	fbSdoReadExUint		:	FB_EcCoESdoReadEx	:= (bCompleteAccess := FALSE);
	fbSdoReadExUdint	:	FB_EcCoESdoReadEx	:= (bCompleteAccess := FALSE);
	fbSdoWriteExSint		:	FB_EcCoESdoWriteEx 	:= (bCompleteAccess := FALSE);
	fbSdoWriteExInt		:	FB_EcCoESdoWriteEx 	:= (bCompleteAccess := FALSE);
	fbSdoWriteExDint		:	FB_EcCoESdoWriteEx 	:= (bCompleteAccess := FALSE);
	fbSdoWriteExUsint	:	FB_EcCoESdoWriteEx 	:= (bCompleteAccess := FALSE);
	fbSdoWriteExUint		:	FB_EcCoESdoWriteEx 	:= (bCompleteAccess := FALSE);
	fbSdoWriteExUdint	:	FB_EcCoESdoWriteEx 	:= (bCompleteAccess := FALSE);
	fbSdoWriteExString	:	FB_EcCoESdoWriteEx 	:= (bCompleteAccess := FALSE);
	fbEcGetSlaveState	:	FB_EcGetSlaveState		;

	fbFileOpen			:	FB_FileOpen				;	(*Used to determine if file exists*)
	fbFileClose			:	FB_FileClose				;	(*Used to determine if file exists*)
END_VAR

fbFallingEdge	(CLK:= bExecute);
IF fbFallingEdge.Q THEN
	bNotExecute	:=	TRUE;
END_IF;

(* Done is TRUE for one cycle when falling edge of Execute has occured *)
IF bDone AND bNotExecute THEN
	bDone		:=	FALSE;
END_IF;

IF bError AND bNotExecute THEN
	bError				:=	FALSE;
	nErrorId				:=	0;
	nErrorIDRead			:=	0;
END_IF;

CASE State OF
0:
fbRisingEdge(CLK:= bExecute);
IF fbRisingEdge.Q THEN
	bDone				:=	FALSE;
	bBusy				:=	TRUE;
	bError				:=	FALSE;
	nErrorId				:=	0;
	nErrorIDRead			:=	0;
	sErrorString			:=	'';
	bNotExecute			:=	FALSE;
	sNetIdRead			:=	sNetId;
	nSlaveAddrRead		:=	nSlaveAddr;
	sFileRead			:=	sFile;
	bBypassCheckRead	:=	bBypassCheck;
	State				:=	1;
	Row					:=	1;
END_IF

1: (*check if file exists by trying to open the file*)
fbFileOpen(
	nMode		:=	FOPEN_MODEREAD,
	sPathName	:=	sFileRead,
	bExecute	:=	TRUE);
State:=2;

2:
fbFileOpen();
IF NOT fbFileOpen.bBusy THEN			(*Check for File Open complete*)
	IF fbFileOpen.bError THEN			(*Check for error from File Open*)
		sErrorString:=CONCAT(CONCAT(
			'Error opening File at  ',
			sFileRead),
			'.  Error occurred using Function Block FB_FileOpen.  ErrorID is from FB_FileOpen.'
		);
		nErrorIDRead:=fbFileOpen.nErrID;
		State:=99;
	ELSE
		fbFileOpen(bExecute := FALSE);
		fbFileClose(
			hFile		:=fbFileOpen.hFile,
			bExecute	:=TRUE);
		State:=3;
	END_IF
END_IF

3:
fbFileClose();
IF NOT fbFileClose.bBusy THEN			(*Check for File Open complete*)
	IF fbFileClose.bError THEN			(*Check for error from File Open*)
		sErrorString:=CONCAT(CONCAT(
			'Error closing File at  ',
			sFileRead),
			'.  Error occurred using Function Block FB_FileClose.  ErrorID is from FB_FileClose.'
		);
		nErrorIDRead:=fbFileOpen.nErrID;
		State:=99;
	ELSE
		fbFileClose(bExecute := FALSE);
		State:=10;
	END_IF
END_IF

10: (*Read Vendor ID from drive*)
fbSdoReadExUdint( 			(*Get Vendor ID*)
	sNetId		:= sNetIdRead,
	nSlaveAddr	:= nSlaveAddrRead ,
	nSubIndex	:= 1,
	nIndex		:= 16#1018,
	pDstBuf		:= ADR(VendorID),
	cbBufLen	:= SIZEOF(VendorID),
	bExecute	:= FALSE 		); (*Rising edge required*)
State:=11;

11: (*running FB for Read Vendor ID*)
fbSdoReadExUdint(bExecute:= TRUE);
State:=12;

12: (*SDO read, Read ID*)
fbSdoReadExUdint();
IF NOT fbSdoReadExUdint.bBusy THEN
	IF NOT fbSdoReadExUdint.bError THEN
		fbSdoReadExUdint(bExecute:= FALSE);
		State:=13;
		IF NOT (VendorID=VENDOR_YASKAWA) THEN 			(*Vendor ID = Yaskawa*)
			sErrorString:=CONCAT(CONCAT(
				'Product not compatible.  This FB is only for Vendor ID 0x00000539 (Yaskawa).  Vendor ID read as ',
				UDINT_TO_STRING(VendorID)),
				'.  ErrorID from FB, not from ADS.'
			);
			nErrorIDRead:=4100;
			State:=99;
		END_IF
	ELSE
		sErrorString:=CONCAT(CONCAT(
			'Error reading Product Code, Object: ',
			WORD_TO_STRING(fbSdoReadExUdint.nIndex)),
			'.  Error occurred using Function Block FB_EcCoESdoReadEx.  ErrorID is from FB_EcCoESdoReadEx.'
		);
		nErrorIDRead:=fbSdoReadExUdint.nErrId;
		State:=99;
	END_IF
END_IF

13:
fbSdoReadExUdint(
	nSubIndex	:= 2,				(*Product Code*)
	pDstBuf		:= ADR(ProductCode),
	cbBufLen	:= SIZEOF(ProductCode),
	bExecute	:= TRUE			);
State:=14;

14: (*Open file to get nID*)
fbSdoReadExUdint();
IF NOT fbSdoReadExUdint.bBusy THEN
	IF NOT fbSdoReadExUdint.bError THEN
		fbFileBuffer.A_Open();
		fbSdoReadExUdint(bExecute:= FALSE);
		State:=15;
		IF ProductCode=PRODUCT_ROTARY THEN 			(*Rotary Motor Detected*)
			AmpType		:= ROTARY;
		ELSE IF ProductCode=PRODUCT_LINEAR THEN 	(*Linear Motor Detected*)
			AmpType		:= LINEAR;
		ELSE 									 (*neither Linear nor Rotary Motor Detected*)
			sErrorString:=CONCAT(CONCAT(
				'Product not compatible.  This FB is only for Product codes 0x02200001 (Sigma-5 Rotary) and 0x02200002 (Sigma-5 Linear).  If using Sigma-5 CoE Drive, get latest FB from Yaskawa.com.  Product code read as ',
				UDINT_TO_STRING(ProductCode)),
				'.  ErrorID from FB, not from ADS.'
			);
			nErrorIDRead:=4101;
			State:=99;
		END_IF
		END_IF
	ELSE
		sErrorString:=CONCAT(CONCAT(
			'Error reading Product Code, Object: ',
			WORD_TO_STRING(fbSdoReadExUdint.nIndex)),
			'.  Error occurred using Function Block FB_EcCoESdoReadEx.  ErrorID is from FB_EcCoESdoReadEx.'
		);
		nErrorIDRead:=fbSdoReadExUdint.nErrId;
		State:=99;
	END_IF
END_IF

15:(*Opened file completed (now can read nID) *)
fbFileBuffer(sPathName:= sFileRead);
IF NOT fbFileBuffer.bBusy THEN									(*Check for File Open complete*)
	IF NOT fbFileBuffer.bError THEN								(*Check for error from File Open*)
		fbSdoReadExUdint(
			nSubIndex	:=3,				(*Revision Number*)
			pDstBuf		:= ADR(RevisionNumber),
			cbBufLen	:= SIZEOF(RevisionNumber),
			bExecute	:= TRUE			);
		State:=16;
	ELSE													(*Error from File Open*)
		sErrorString:=CONCAT(CONCAT(
			'Error opening File at  ',
			sFileRead),
			'.  Error occurred using Function Call FB_FileRingBuffer.A_Open.  ErrorID is from FB_FileRingBuffer.'
		);
		nErrorIDRead:=fbFileBuffer.nErrID;
		State:=99;
	END_IF
END_IF

16: (*Check Revision Number and check file created by a Function Block version*)
fbSdoReadExUdint();
IF NOT fbSdoReadExUdint.bBusy THEN
	IF NOT fbSdoReadExUdint.bError THEN
		IF RevisionNumber=REVISION_1
(*Vers Up*)	OR RevisionNumber=REVISION_2
			OR bBypassCheckRead
			THEN 		(*Version 1.0, 2.0*) (*IF statement to allow future version implementations*)
			IF fbFileBuffer.stHeader.nID=Y_FB_VER_1_0
(*Vers Up*)		OR fbFileBuffer.stHeader.nID=Y_FB_VER_2_0
				THEN
				fbSdoReadExUdint(bExecute:= FALSE);
				fbFileBuffer.A_GetHead(				(*Read from open file*)
					pReadBuff	:= ADR(AllSigmaObjects),
					cbReadLen	:= SIZEOF(AllSigmaObjects));
				State:=17;
			ELSE IF fbFileBuffer.stHeader.status.1=1 THEN
					sErrorString:='File is corrupt.  Store the parameters again. ErrorID from FB, not from ADS';
					nErrorIDRead:=4104;
					State:=99;
				ELSE IF fbFileBuffer.stHeader.nID=0 THEN
					sErrorString:='No version of ID of file was read.  Possibly incorrect file, or FB has an error. ErrorID from FB, not from ADS.';
					nErrorIDRead:=4105;
					State:=99;
				ELSE
					sErrorString:=CONCAT(CONCAT(CONCAT(CONCAT(
						'This file was made with a different version than this Function Block. Obtain the latest FB from Yaskawa.com.  Current FB version is ',
						UDINT_TO_STRING(FbVersion)),
						 '.  File version is '),
						UDINT_TO_STRING(fbFileBuffer.stHeader.nID)),
						'.  ErrorID from FB, not from ADS.'
					);
					nErrorIDRead:=4106;
					State:=99;
				END_IF
				END_IF
			END_IF
		ELSE 									 (*Incorrect version used*)
			sErrorString:=CONCAT(CONCAT(
(*Vers Up*)		'Product not compatible.  This FB is only for Revision Number 0x00010000 (Vers.1.0) and 0x00020000 (Vers.2.0).  If using Sigma-5 CoE Drive, get latest FB from Yaskawa.com.  Revision Number read as ',
				UDINT_TO_STRING(RevisionNumber)),
				'.  ErrorID from FB, not from ADS.'
			);
			nErrorIDRead:=4102;
			State:=99;
		END_IF
	ELSE
		sErrorString:=CONCAT(CONCAT(
			'Error reading Product Code, Object: ',
			WORD_TO_STRING(fbSdoReadExUdint.nIndex)),
			'.  Error occurred using Function Block FB_EcCoESdoReadEx.  ErrorID is from FB_EcCoESdoReadEx.'
		);
		nErrorIDRead:=fbSdoReadExUdint.nErrId;
		State:=99;
	END_IF
END_IF

17:
fbFileBuffer();
IF NOT fbFileBuffer.bBusy THEN
	IF NOT fbFileBuffer.bError THEN
		fbFileBuffer.A_Close();
		State:=20;
	ELSE
		sErrorString:=CONCAT(CONCAT(
			'Error reading Sigma Object Data from ',
			sFileRead),
			'.  Error occurred with function call FB_FileRingBuffer.A_GetHead.  ErrorID is from FB_FileRingBuffer.'
		);
		nErrorIDRead:=fbFileBuffer.nErrID;
		State:=99;
	END_IF
END_IF

20: (*File closed, check for FSA state "Swich On Disabled"*)
fbFileBuffer();
IF NOT fbFileBuffer.bBusy THEN
	IF NOT fbFileBuffer.bError THEN
		State:=21;
		fbSdoReadExUint( 			(*Get StatusWord*)
			sNetId		:= sNetIdRead,
			nSlaveAddr	:= nSlaveAddrRead ,
			nSubIndex	:= 0,
			nIndex		:= 16#6041,
			pDstBuf		:= ADR(StatusWord),
			cbBufLen	:= SIZEOF(StatusWord),
			bExecute	:= FALSE 		); (*rising edge required*)
	ELSE
		sErrorString:=CONCAT(CONCAT(
			'Error closing re-created file: ',
			sFileRead),
			'.  Error occurred using Function Call FB_FileRingBuffer.A_Close.  ErrorID is from FB_FileRingBuffer.'
		);
		nErrorIDRead:=fbFileBuffer.nErrID;
		State:=99;
	END_IF
END_IF

21:
fbSdoReadExUint(bExecute := TRUE);
State:=22;

22:
fbSdoReadExUint();
IF NOT fbSdoReadExUint.bBusy THEN
	IF NOT fbSdoReadExUint.bError THEN
		fbSdoReadExUint(bExecute:= FALSE);
		IF (UINT_TO_WORD(StatusWord) AND 2#0000_0000_0100_1111)=2#0000_0000_0100_0000 THEN 	(*"switch on disabled" state*)
			fbEcGetSlaveState( (*Writing parameters require PRE-OP.*)
				sNetId		:= sNetIdRead,
				nSlaveAddr	:= nSlaveAddrRead ,
				bExecute	:= FALSE 		); (*rising edge required*)
			State:=23;
		ELSE
			sErrorString:=CONCAT(CONCAT(
				'Not in FSA state Swich On Disabled.  StatusWord expected as x1xx_0000 (bin), but read as ',
				UDINT_TO_STRING(StatusWord)),
				'(dec).  ErrorID from FB, not from ADS.'
			);
			nErrorIDRead:=4107;
			State:=99;
		END_IF
	ELSE
		sErrorString:=CONCAT(CONCAT(
			'Error reading StatusWord, Object: ',
			WORD_TO_STRING(fbSdoReadExUint.nIndex)),
			'.  Error occurred using Function Block FB_EcCoESdoReadEx.  ErrorID is from FB_EcCoESdoReadEx.'
		);
		nErrorIDRead:=fbSdoReadExUint.nErrId;
		State:=99;
	END_IF
END_IF

23:
fbEcGetSlaveState(bExecute := TRUE);
State:=24;

24:
fbEcGetSlaveState();
IF NOT fbEcGetSlaveState.bBusy THEN
	IF NOT fbEcGetSlaveState.bError THEN
		fbEcGetSlaveState(bExecute:= FALSE);
		IF fbEcGetSlaveState.state.deviceState=EC_DEVICE_STATE_PREOP THEN
			fbSdoWriteExSint(
				sNetId		:= sNetIdRead,
				nSlaveAddr	:= nSlaveAddrRead,
				bExecute	:= FALSE			);
			fbSdoWriteExInt(
				sNetId		:= sNetIdRead,
				nSlaveAddr	:= nSlaveAddrRead,
				bExecute	:= FALSE			);
			fbSdoWriteExDint(
				sNetId		:= sNetIdRead,
				nSlaveAddr	:= nSlaveAddrRead,
				bExecute	:= FALSE			);
			fbSdoWriteExUsint(
				sNetId		:= sNetIdRead,
				nSlaveAddr	:= nSlaveAddrRead,
				bExecute	:= FALSE			);
			fbSdoWriteExUint(
				sNetId		:= sNetIdRead,
				nSlaveAddr	:= nSlaveAddrRead,
				bExecute	:= FALSE			);
			fbSdoWriteExUdint(
				sNetId		:= sNetIdRead,
				nSlaveAddr	:= nSlaveAddrRead,
				bExecute	:= FALSE			);
			fbSdoWriteExString(
				sNetId		:= sNetIdRead,
				nSlaveAddr	:= nSlaveAddrRead,
				bExecute	:= FALSE			);
			State:=30;
		ELSE
			sErrorString:=CONCAT(CONCAT(
				'Drive not set to PRE-OP mode.  Set the drive to PRE-OP mode before using this FB.  Enumerated mode read as: ',
				BYTE_TO_STRING(fbEcGetSlaveState.state.deviceState)),
				'.  ErrorID is custom for this FB.'
				);
			nErrorIDRead:=4108;
			State:=99;
		END_IF
	ELSE
		sErrorString:='Error reading Slave State.  Error occurred using Function Block FB_EcGetSlaveState.  ErrorID is from FB_EcGetSlaveState.';
		nErrorIDRead:=fbEcGetSlaveState.nErrId;
		State:=99;
	END_IF
END_IF

30: (*now in preop, write DEPENDENT pre-op parameters, (those that conditional prms depend on)*)
IF NOT (Row=MaxRows+1) THEN
	IF
		(AllSigmaObjects[Row].AmpType=BOTH_ROT_LIN	(*If parameter set is for either rotary/linear*)
		OR AllSigmaObjects[Row].AmpType=AmpType)		(*parameter set is for just rotary or just linear*)
		AND AllSigmaObjects[Row].Access=ACCESS_RW		(*Parameter has RW access*)
		AND NOT ((AllSigmaObjects[Row].SpecialParameter AND INT_TO_WORD(OBJECT_COMMAND))	=INT_TO_WORD(OBJECT_COMMAND))
		AND ((AllSigmaObjects[Row].SpecialParameter AND INT_TO_WORD(HAS_DEPENDENT))			=INT_TO_WORD(HAS_DEPENDENT))
	THEN
		CASE AllSigmaObjects[Row].ValueType OF
		TYPE_USINT:
			fbSdoWriteExUsint(
				nIndex		:= AllSigmaObjects[Row].Index,
				nSubIndex	:= AllSigmaObjects[Row].SubIndex,
				pSrcBuf		:= ADR(AllSigmaObjects[Row].DependentValueUsint),
				cbBufLen	:= SIZEOF(AllSigmaObjects[Row].DependentValueUsint),
				bExecute	:= TRUE );
			State:=40;
		ELSE
			sErrorString:=CONCAT(CONCAT(
				'Error reading Object Data Type or Data Type not supported.  Enumerated value read as: ',
				USINT_TO_STRING(AllSigmaObjects[Row].ValueType)),
				'.'
			);
			nErrorIDRead:=4103;
			State:=99;
		END_CASE
	ELSE
		Row:=Row+1;
	END_IF
ELSE
	Row:=1;
	State:=100;
END_IF

40:
fbSdoWriteExUsint();
IF NOT fbSdoWriteExUsint.bBusy THEN (*extra check just in case*)
	IF NOT fbSdoWriteExUsint.bError THEN
		Row:=Row+1;
		fbSdoWriteExUsint(bExecute:= FALSE);
		State:=30;
	ELSE
		sErrorString:=CONCAT(CONCAT(
			'Error writing CoE Object ',
			WORD_TO_STRING(AllSigmaObjects[Row].Index)),
			'.  Error occurred using Function Block FB_EcCoESdoWriteEx.  ErrorID is from FB_EcCoESdoWriteEx.'
		);
		nErrorIDRead:=fbSdoWriteExUsint.nErrId;
		State:=99;
	END_IF
END_IF

100: (*write the HAS_DEPENDENTs first*)
IF NOT (Row=MaxRows+1) THEN
	IF
		(AllSigmaObjects[Row].AmpType=BOTH_ROT_LIN	(*If parameter set is for either rotary/linear*)
		OR AllSigmaObjects[Row].AmpType=AmpType)		(*parameter set is for just rotary or just linear*)
		AND AllSigmaObjects[Row].Access=ACCESS_RW		(*Parameter has RW access*)
		AND NOT ((AllSigmaObjects[Row].SpecialParameter AND INT_TO_WORD(OBJECT_COMMAND))		=INT_TO_WORD(OBJECT_COMMAND))
		AND NOT ((AllSigmaObjects[Row].SpecialParameter AND INT_TO_WORD(HAS_DEPENDENT))			=INT_TO_WORD(HAS_DEPENDENT))
	THEN
		CASE AllSigmaObjects[Row].ValueType OF
		TYPE_SINT:
			fbSdoWriteExSint(
				nIndex		:= AllSigmaObjects[Row].Index,
				nSubIndex	:= AllSigmaObjects[Row].SubIndex,
				pSrcBuf		:= ADR(AllSigmaObjects[Row].ValueSint),
				cbBufLen	:= SIZEOF(AllSigmaObjects[Row].ValueSint),
				bExecute	:= TRUE );
			State:=120;
		TYPE_INT:
			fbSdoWriteExInt(
				nIndex		:= AllSigmaObjects[Row].Index,
				nSubIndex	:= AllSigmaObjects[Row].SubIndex,
				pSrcBuf		:= ADR(AllSigmaObjects[Row].ValueInt),
				cbBufLen	:= SIZEOF(AllSigmaObjects[Row].ValueInt),
				bExecute	:= TRUE );
			State:=130;
		TYPE_DINT:
			fbSdoWriteExDint(
				nIndex		:= AllSigmaObjects[Row].Index,
				nSubIndex	:= AllSigmaObjects[Row].SubIndex,
				pSrcBuf		:= ADR(AllSigmaObjects[Row].ValueDint),
				cbBufLen	:= SIZEOF(AllSigmaObjects[Row].ValueDint),
				bExecute	:= TRUE );
			State:=140;
		TYPE_USINT:
			fbSdoWriteExUsint(
				nIndex		:= AllSigmaObjects[Row].Index,
				nSubIndex	:= AllSigmaObjects[Row].SubIndex,
				pSrcBuf		:= ADR(AllSigmaObjects[Row].ValueUsint),
				cbBufLen	:= SIZEOF(AllSigmaObjects[Row].ValueUsint),
				bExecute	:= TRUE );
			State:=150;
		TYPE_UINT:
			fbSdoWriteExUint(
				nIndex		:= AllSigmaObjects[Row].Index,
				nSubIndex	:= AllSigmaObjects[Row].SubIndex,
				pSrcBuf		:= ADR(AllSigmaObjects[Row].ValueUint),
				cbBufLen	:= SIZEOF(AllSigmaObjects[Row].ValueUint),
				bExecute	:= TRUE );
			State:=160;
		TYPE_UDINT:
			fbSdoWriteExUdint(
				nIndex		:= AllSigmaObjects[Row].Index,
				nSubIndex	:= AllSigmaObjects[Row].SubIndex,
				pSrcBuf		:= ADR(AllSigmaObjects[Row].ValueUdint),
				cbBufLen	:= SIZEOF(AllSigmaObjects[Row].ValueUdint),
				bExecute	:= TRUE );
			State:=170;
		TYPE_STRING:
			fbSdoWriteExString(
				nIndex		:= AllSigmaObjects[Row].Index,
				nSubIndex	:= AllSigmaObjects[Row].SubIndex,
				pSrcBuf		:= ADR(AllSigmaObjects[Row].ValueString),
				cbBufLen	:= SIZEOF(AllSigmaObjects[Row].ValueString),
				bExecute	:= TRUE );
			State:=180;
		ELSE
			sErrorString:=CONCAT(CONCAT(
				'Error reading Object Data Type or Data Type not supported.  Enumerated value read as: ',
				USINT_TO_STRING(AllSigmaObjects[Row].ValueType)),
				'.'
			);
			nErrorIDRead:=4103;
			State:=99;
		END_CASE
	
	ELSE
		Row:=Row+1;
	END_IF
ELSE
	Row:=1;
	State:=200;
END_IF

120:
fbSdoWriteExSint();
IF NOT fbSdoWriteExSint.bBusy THEN (*extra check just in case*)
	IF NOT fbSdoWriteExSint.bError THEN
		Row:=Row+1;
		fbSdoWriteExSint(bExecute:= FALSE);
		State:=100;
	ELSE
		sErrorString:=CONCAT(CONCAT(
			'Error writing CoE Object  ',
			WORD_TO_STRING(AllSigmaObjects[Row].Index)),
			'.  Error occurred using Function Block FB_EcCoESdoWriteEx.  ErrorID is from FB_EcCoESdoWriteEx.'
		);
		nErrorIDRead:=fbSdoWriteExSint.nErrId;
		State:=99;
	END_IF
END_IF

130:
fbSdoWriteExInt();
IF NOT fbSdoWriteExInt.bBusy THEN (*extra check just in case*)
	IF NOT fbSdoWriteExInt.bError THEN
		Row:=Row+1;
		fbSdoWriteExInt(bExecute:= FALSE);
		State:=100;
	ELSE
		sErrorString:=CONCAT(CONCAT(
			'Error writing CoE Object ',
			WORD_TO_STRING(AllSigmaObjects[Row].Index)),
			'.  Error occurred using Function Block FB_EcCoESdoWriteEx.  ErrorID is from FB_EcCoESdoWriteEx.'
		);
		nErrorIDRead:=fbSdoWriteExInt.nErrId;
		State:=99;
	END_IF
END_IF

140:
fbSdoWriteExDint();
IF NOT fbSdoWriteExDint.bBusy THEN (*extra check just in case*)
	IF NOT fbSdoWriteExDint.bError THEN
		Row:=Row+1;
		fbSdoWriteExDint(bExecute:= FALSE);
		State:=100;
	ELSE
		sErrorString:=CONCAT(CONCAT(
			'Error writing CoE Object ',
			WORD_TO_STRING(AllSigmaObjects[Row].Index)),
			'.  Error occurred using Function Block FB_EcCoESdoWriteEx.  ErrorID is from FB_EcCoESdoWriteEx.'
		);
		nErrorIDRead:=fbSdoWriteExDint.nErrId;
		State:=99;
	END_IF
END_IF

150:
fbSdoWriteExUsint();
IF NOT fbSdoWriteExUsint.bBusy THEN (*extra check just in case*)
	IF NOT fbSdoWriteExUsint.bError THEN
		Row:=Row+1;
		fbSdoWriteExUsint(bExecute:= FALSE);
		State:=100;
	ELSE
		sErrorString:=CONCAT(CONCAT(
			'Error writing CoE Object ',
			WORD_TO_STRING(AllSigmaObjects[Row].Index)),
			'.  Error occurred using Function Block FB_EcCoESdoWriteEx.  ErrorID is from FB_EcCoESdoWriteEx.'
		);
		nErrorIDRead:=fbSdoWriteExUsint.nErrId;
		State:=99;
	END_IF
END_IF

160:
fbSdoWriteExUint();
IF NOT fbSdoWriteExUint.bBusy THEN (*extra check just in case*)
	IF NOT fbSdoWriteExUint.bError THEN
		Row:=Row+1;
		fbSdoWriteExUint(bExecute:= FALSE);
		State:=100;
	ELSE
		sErrorString:=CONCAT(CONCAT(
			'Error writing CoE Object ',
			WORD_TO_STRING(AllSigmaObjects[Row].Index)),
			'.  Error occurred using Function Block FB_EcCoESdoWriteEx.  ErrorID is from FB_EcCoESdoWriteEx.'
		);
		nErrorIDRead:=fbSdoWriteExUint.nErrId;
		State:=99;
	END_IF
END_IF

170:
fbSdoWriteExUdint();
IF NOT fbSdoWriteExUdint.bBusy THEN (*extra check just in case*)
	IF NOT fbSdoWriteExUdint.bError THEN
		Row:=Row+1;
		fbSdoWriteExUdint(bExecute:= FALSE);
		State:=100;
	ELSE
		sErrorString:=CONCAT(CONCAT(
			'Error writing CoE Object ',
			WORD_TO_STRING(AllSigmaObjects[Row].Index)),
			'.  Error occurred using Function Block FB_EcCoESdoWriteEx.  ErrorID is from FB_EcCoESdoWriteEx.'
		);
		nErrorIDRead:=fbSdoWriteExUdint.nErrId;
		State:=99;
	END_IF
END_IF

180:
fbSdoWriteExString();
IF NOT fbSdoWriteExString.bBusy THEN (*extra check just in case*)
	IF NOT fbSdoWriteExString.bError THEN
		Row:=Row+1;
		fbSdoWriteExString(bExecute:= FALSE);
		State:=100;
	ELSE
		sErrorString:=CONCAT(CONCAT(
			'Error writing CoE Object ',
			WORD_TO_STRING(AllSigmaObjects[Row].Index)),
			'.  Error occurred using Function Block FB_EcCoESdoWriteEx.  ErrorID is from FB_EcCoESdoWriteEx.'
		);
		nErrorIDRead:=fbSdoWriteExString.nErrId;
		State:=99;
	END_IF
END_IF

200: (*Written prms in pre-op, now need to set HAS_DEPENDENT prms from saved prm file*)
IF NOT (Row=MaxRows+1) THEN
	IF
		(AllSigmaObjects[Row].AmpType=BOTH_ROT_LIN	(*If parameter set is for either rotary/linear*)
		OR AllSigmaObjects[Row].AmpType=AmpType)		(*parameter set is for just rotary or just linear*)
		AND AllSigmaObjects[Row].Access=ACCESS_RW		(*Parameter has RW access*)
		AND NOT ((AllSigmaObjects[Row].SpecialParameter AND INT_TO_WORD(OBJECT_COMMAND))	=INT_TO_WORD(OBJECT_COMMAND))
		AND ((AllSigmaObjects[Row].SpecialParameter AND INT_TO_WORD(HAS_DEPENDENT))			=INT_TO_WORD(HAS_DEPENDENT))

	THEN
		CASE AllSigmaObjects[Row].ValueType OF
		TYPE_USINT:
			fbSdoWriteExUsint(
				nIndex		:= AllSigmaObjects[Row].Index,
				nSubIndex	:= AllSigmaObjects[Row].SubIndex,
				pSrcBuf		:= ADR(AllSigmaObjects[Row].ValueUsint),
				cbBufLen	:= SIZEOF(AllSigmaObjects[Row].ValueUsint),
				bExecute	:= TRUE );
			State:=210;
		ELSE
			sErrorString:=CONCAT(CONCAT(
				'Error reading Object Data Type or Data Type not supported.  Enumerated value read as: ',
				USINT_TO_STRING(AllSigmaObjects[Row].ValueType)),
				'.'
			);
			nErrorIDRead:=4103;
			State:=99;
		END_CASE
	ELSE
		Row:=Row+1;
	END_IF
ELSE
	Row:=1;
	State:=300;
END_IF

210:
fbSdoWriteExUsint();
IF NOT fbSdoWriteExUsint.bBusy THEN (*extra check just in case*)
	IF NOT fbSdoWriteExUsint.bError THEN
		Row:=Row+1;
		fbSdoWriteExUsint(bExecute:= FALSE);
		State:=200;
	ELSE
		sErrorString:=CONCAT(CONCAT(
			'Error writing CoE Object ',
			WORD_TO_STRING(AllSigmaObjects[Row].Index)),
			'.  Error occurred using Function Block FB_EcCoESdoWriteEx.  ErrorID is from FB_EcCoESdoWriteEx.'
		);
		nErrorIDRead:=fbSdoWriteExUsint.nErrId;
		State:=99;
	END_IF
END_IF

300:
fbSdoWriteExUdint(
	nIndex		:= 16#1010,
	nSubIndex	:= 1,
	pSrcBuf		:= ADR(SAVE),
	cbBufLen	:= SIZEOF(SAVE),
	bExecute	:= TRUE );
State:=301;

301:
fbSdoWriteExUdint();
IF NOT fbSdoWriteExUdint.bBusy THEN (*extra check just in case*)
	IF NOT fbSdoWriteExUdint.bError THEN
		fbSdoWriteExUdint(bExecute:= FALSE);
		State:=302;
	ELSE
		sErrorString:=CONCAT(CONCAT(
			'Error writing CoE Object ',
			WORD_TO_STRING(fbSdoWriteExUdint.nIndex)),
			'.  Error occurred using Function Block FB_EcCoESdoWriteEx.  ErrorID is from FB_EcCoESdoWriteEx.'
		);
		nErrorIDRead:=fbSdoWriteExUdint.nErrId;
		State:=99;
	END_IF
END_IF

302:
fbSdoReadExUdint(
	nIndex		:= 16#1010,
	nSubIndex	:= 1,
	pDstBuf		:= ADR(StorePrmStatus),
	cbBufLen	:= SIZEOF(StorePrmStatus),
	bExecute	:= TRUE			);
State:=303;

303:
fbSdoReadExUdint();
IF NOT fbSdoReadExUdint.bBusy THEN
	IF NOT fbSdoReadExUdint.bError THEN
		fbSdoReadExUdint(bExecute:= FALSE);
		IF StorePrmStatus=1THEN
			State:=304;
		ELSE
			State:=302;
		END_IF
	ELSE
		sErrorString:=CONCAT(CONCAT(
			'Error reading Save Parameter, Object: ',
			WORD_TO_STRING(fbSdoReadExUdint.nIndex)),
			'.  Error occurred using Function Block FB_EcCoESdoReadEx.  ErrorID is from FB_EcCoESdoReadEx.'
		);
		nErrorIDRead:=fbSdoReadExUdint.nErrId;
		State:=99;
	END_IF
END_IF

304:
fbSdoWriteExUdint(
	nIndex		:= 16#2700,
	nSubIndex	:= 0,
	pSrcBuf		:= ADR(USERPRMCFG),
	cbBufLen	:= SIZEOF(USERPRMCFG),
	bExecute	:= TRUE );
State:=305;

305:
fbSdoWriteExUdint();
IF NOT fbSdoWriteExUdint.bBusy THEN (*extra check just in case*)
	IF NOT fbSdoWriteExUdint.bError THEN
		fbSdoWriteExUdint(bExecute:= FALSE);
		State:=306;
	ELSE
		sErrorString:=CONCAT(CONCAT(
			'Error writing CoE Object ',
			WORD_TO_STRING(fbSdoWriteExUdint.nIndex)),
			'.  Error occurred using Function Block FB_EcCoESdoWriteEx.  ErrorID is from FB_EcCoESdoWriteEx.'
		);
		nErrorIDRead:=fbSdoWriteExUdint.nErrId;
		State:=99;
	END_IF
END_IF

306:
fbSdoReadExUdint(
	nIndex		:= 16#2700,
	nSubIndex	:= 0,
	pDstBuf		:= ADR(PrmCfgStatus),
	cbBufLen	:= SIZEOF(PrmCfgStatus),
	bExecute	:= TRUE			);
State:=307;

307:
fbSdoReadExUdint();
IF NOT fbSdoReadExUdint.bBusy THEN
	IF NOT fbSdoReadExUdint.bError THEN
		fbSdoReadExUdint(bExecute:= FALSE);
		IF PrmCfgStatus=0THEN
			bDone	:=	TRUE;
			bBusy	:=	FALSE;
			State:=0;
		ELSE
			State:=306;
		END_IF
	ELSE
		sErrorString:=CONCAT(CONCAT(
			'Error reading User Parameter Config, Object: ',
			WORD_TO_STRING(fbSdoReadExUdint.nIndex)),
			'.  Error occurred using Function Block FB_EcCoESdoReadEx.  ErrorID is from FB_EcCoESdoReadEx.'
		);
		nErrorIDRead:=fbSdoReadExUdint.nErrId;
		State:=99;
	END_IF
END_IF

99: (*Error State*)
	bBusy	:=	FALSE;
	bError	:=	TRUE;
	nErrorID	:=	nErrorIDRead;
	State	:=	0;
ELSE
;
END_CASE

END_FUNCTION_BLOCK
